Staubli VAL3: JPOINT.dtx

public TrajJoint tTraj{}
  [cuigan1]
    num nIndexFrame
    num nIndexTool
    string sID = "cuigan1"
    TrajJointItem tData[4]
      [0]
        jointRx jJoint = {j1=43.073741, j2=-21.440622, j3=-75.766984, j4=-1.055518, j5=-80.962605, j6=-104.91072}
        TrajectoryItem tSuper
          [0]
            string comment
            num distance
            InstrItem iInstr[3]
              [0]
                string sData
                string sType
              [1]
                string sData
                string sType
              [2]
                string sData
                string sType
            num moveType
            num nMoveId
            num nStop
            num nTcpAction
            num nTime
            mdesc nom_speed = {tmax=9999}
            bool toStop
      [1]
        jointRx jJoint = {j1=22.638661, j2=-19.809054, j3=-65.603625, j4=-1.089653, j5=-90.904739, j6=-104.362244}
        TrajectoryItem tSuper
          [0]
            string comment
            num distance
            InstrItem iInstr[3]
              [0]
                string sData
                string sType
              [1]
                string sData
                string sType
              [2]
                string sData
                string sType
            num moveType
            num nMoveId
            num nStop
            num nTcpAction
            num nTime
            mdesc nom_speed = {tmax=9999}
            bool toStop
      [2]
        jointRx jJoint = {j1=-65.330843, j2=-19.809054, j3=-65.603625, j4=-1.089653, j5=-90.904739, j6=-104.362244}
        TrajectoryItem tSuper
          [0]
            string comment
            num distance
            InstrItem iInstr[3]
              [0]
                string sData
                string sType
              [1]
                string sData
                string sType
              [2]
                string sData
                string sType
            num moveType
            num nMoveId
            num nStop
            num nTcpAction
            num nTime
            mdesc nom_speed = {tmax=9999}
            bool toStop
      [3]
        jointRx jJoint = {j1=-47.626065, j2=-20.138594, j3=-86.728564, j4=-0.126452, j5=-74.274403, j6=-229.27512}
        TrajectoryItem tSuper
          [0]
            string comment
            num distance
            InstrItem iInstr[3]
              [0]
                string sData
                string sType
              [1]
                string sData
                string sType
              [2]
                string sData
                string sType
            num moveType
            num nMoveId
            num nStop
            num nTcpAction
            num nTime
            mdesc nom_speed = {tmax=9999}
            bool toStop
  [cuigan2]
    num nIndexFrame
    num nIndexTool
    string sID = "cuigan2"
    TrajJointItem tData[3]
      [0]
        jointRx jJoint = {j1=-46.369517, j2=-34.132644, j3=-102.583351, j4=-130.640502, j5=-58.847287, j6=56.297342}
        TrajectoryItem tSuper
          [0]
            string comment
            num distance
            InstrItem iInstr[3]
              [0]
                string sData
                string sType
              [1]
                string sData
                string sType
              [2]
                string sData
                string sType
            num moveType
            num nMoveId
            num nStop
            num nTcpAction
            num nTime
            mdesc nom_speed = {tmax=9999}
            bool toStop
      [1]
        jointRx jJoint = {j1=-77.711525, j2=-21.244592, j3=-128.557253, j4=-169.471735, j5=-60.542274, j6=82.373524}
        TrajectoryItem tSuper
          [0]
            string comment
            num distance
            InstrItem iInstr[3]
              [0]
                string sData
                string sType
              [1]
                string sData
                string sType
              [2]
                string sData
                string sType
            num moveType
            num nMoveId
            num nStop
            num nTcpAction
            num nTime
            mdesc nom_speed = {tmax=9999}
            bool toStop
      [2]
        jointRx jJoint = {j1=-96.007162, j2=-51.391769, j3=-129.725703, j4=-189.143372, j5=-91.420326, j6=87.469449}
        TrajectoryItem tSuper
          [0]
            string comment
            num distance
            InstrItem iInstr[3]
              [0]
                string sData
                string sType
              [1]
                string sData
                string sType
              [2]
                string sData
                string sType
            num moveType
            num nMoveId
            num nStop
            num nTcpAction
            num nTime
            mdesc nom_speed = {tmax=9999}
            bool toStop
  [huilu]
    num nIndexFrame
    num nIndexTool
    string sID = "huilu"
    TrajJointItem tData[5]
      [0]
        jointRx jJoint = {j1=-100.5129, j2=2.60797, j3=-87.026172, j4=-181.161846, j5=94.86685, j6=79.804247}
        TrajectoryItem tSuper
          [0]
            string comment
            num distance
            InstrItem iInstr[3]
              [0]
                string sData
                string sType
              [1]
                string sData
                string sType
              [2]
                string sData
                string sType
            num moveType
            num nMoveId
            num nStop
            num nTcpAction
            num nTime
            mdesc nom_speed = {tmax=9999, blend=off}
            bool toStop
      [1]
        jointRx jJoint = {j1=78.348626, j2=-8.951665, j3=-74.704253, j4=-181.198003, j5=95.687826, j6=-99.806363}
        TrajectoryItem tSuper
          [0]
            string comment
            num distance
            InstrItem iInstr[3]
              [0]
                string sData
                string sType
              [1]
                string sData
                string sType
              [2]
                string sData
                string sType
            num moveType
            num nMoveId
            num nStop
            num nTcpAction
            num nTime
            mdesc nom_speed = {tmax=9999, blend=off}
            bool toStop
      [2]
        jointRx jJoint = {j1=89.491746, j2=17.962399, j3=-111.372053, j4=-181.198003, j5=-0.634174, j6=-89.448803}
        TrajectoryItem tSuper
          [0]
            string comment
            num distance
            InstrItem iInstr[3]
              [0]
                string sData
                string sType
              [1]
                string sData
                string sType
              [2]
                string sData
                string sType
            num moveType
            num nMoveId
            num nStop
            num nTcpAction
            num nTime
            mdesc nom_speed = {tmax=9999, blend=off}
            bool toStop
      [3]
        jointRx jJoint = {j1=89.750307, j2=-11.492067, j3=-121.919508, j4=-179.624051, j5=-40.635948, j6=-90.919459}
        TrajectoryItem tSuper
          [0]
            string comment
            num distance
            InstrItem iInstr[3]
              [0]
                string sData
                string sType
              [1]
                string sData
                string sType
              [2]
                string sData
                string sType
            num moveType
            num nMoveId
            num nStop
            num nTcpAction
            num nTime
            mdesc nom_speed = {tmax=9999, blend=off}
            bool toStop
      [4]
        jointRx jJoint = {j1=89.750339, j2=-61.16853, j3=-123.267439, j4=-179.754871, j5=-91.659213, j6=-90.62711}
        TrajectoryItem tSuper
          [0]
            string comment
            num distance
            InstrItem iInstr[3]
              [0]
                string sData
                string sType
              [1]
                string sData
                string sType
              [2]
                string sData
                string sType
            num moveType
            num nMoveId
            num nStop
            num nTcpAction
            num nTime
            mdesc nom_speed = {tmax=9999, blend=off}
            bool toStop
